TYPE ST_Contactor :
STRUCT
    bCmd      : BOOL;
    bTakeCtrl : BOOL;
    bOut      : BOOL;
END_STRUCT
END_TYPE

(* stored: Version 1.1.0.1, ProductVersion 3.1.4024.16
   DUT ST_Contactor: Id {d7069320-8af6-452a-a94f-be13ae1514da} *)
